FUNCTION_BLOCK Sequence4
VAR_INPUT
END_VAR
VAR_OUTPUT
END_VAR
VAR
END_VAR

END_FUNCTION_BLOCK

(* stored: Version 1.1.0.1, ProductVersion 3.1.4024.11
   POU Sequence4: Id {2f457965-dc86-4899-85e2-e131921b13d1}, SpecialFunc None *)
